Fanuc KAREL source: kb00087.KL

-- PROVISIONAL review KL for V1013-1; original PC SHA256 441274c7c8db640fba0177293ac94e9ef7be4e617d10d4fe04e7643a1f1fa989
-- Incomplete behavior may be omitted. Consult companion uncertainty JSON. Do not deploy.
PROGRAM KB00087
%NOLOCKGROUP
BEGIN
  -- UNRESOLVED_PC offsets 5-12; opcodes 9D,23
  -- UNRESOLVED_PC offsets 17-24; opcodes 9D,23
  -- UNRESOLVED_PC offsets 29-59; opcodes 27,22,22,27,9D,31,7E,4A
  -- UNRESOLVED_PC offsets 64-68; opcodes 7F
END KB00087
